ABB RAPID module: DecorationMovementV3

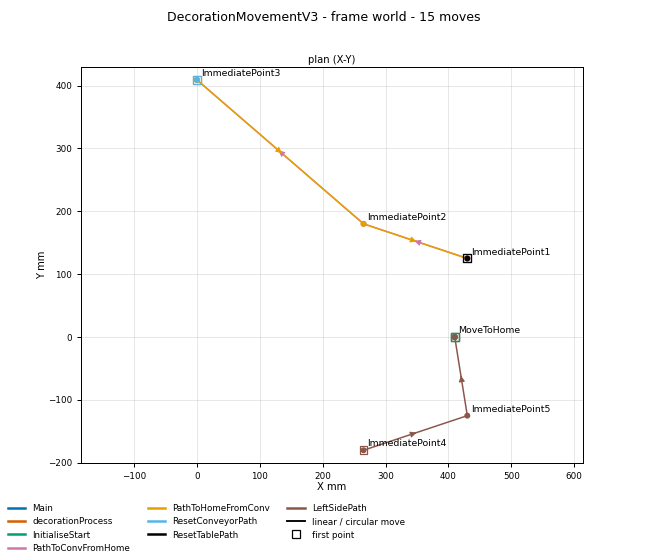
[picture p0: tool path of DecorationMovementV3 in frame world, 15 of 19 moves have a stored position in this frame; points joined in program order, loops and branches not executed]
MODULE DecorationFinal
!***************************************************************
! Decoration Movement Code for Robot
! Author: Dylan Dam z5115759
!***************************************************************


    ! Custom waypoints that I have selected
    CONST robtarget ImmediatePoint1:=[[430,125,450],[0,0,1,0],[0,-1,0,0],[9E+09,9E+09,9E+09,9E+09,9E+09,9E+09]];
    CONST robtarget ImmediatePoint2:=[[265,180,450],[0,0,1,0],[0,-1,0,0],[9E+09,9E+09,9E+09,9E+09,9E+09,9E+09]];
    CONST robtarget ImmediatePoint3:=[[0,409,450],[0,0,1,0],[1,-1,1,0],[9E+09,9E+09,9E+09,9E+09,9E+09,9E+09]];
    CONST robtarget ImmediatePoint4:=[[265,-180,450],[0,0,1,0],[1,-1,1,0],[9E+09,9E+09,9E+09,9E+09,9E+09,9E+09]];
    CONST robtarget ImmediatePoint5:=[[430,-125,450],[0,0,1,0],[1,-1,1,0],[9E+09,9E+09,9E+09,9E+09,9E+09,9E+09]];
    CONST robtarget MoveToHome:=[[410,0,450],[0,0,-1,0],[0,0,-1,0],[9E+09,9E+09,9E+09,9E+09,9E+09,9E+09]];
    ! Offset for the end-effector
    CONST num offSet := 75;
    !Dummy Array for Testing
    !CONST num qwirkleArray{4,7} := [[0,409,22.1,175,0,147,45],[0,409,22.1,548.6,0,147,0],[0,409,22.1,175,520,147,-45],[0,409,22.1,175,-300,147,-45]];
    CONST num qwirkleArray{1,7} := [[0,409,22.1,175,-50,147,-89]];

    PROC Main()
        MoveL MoveToHome,v1000,z100,tool0\WObj:=wobj0;
        decorationProcess qwirkleArray;
        MoveL MoveToHome,v1000,z100,tool0\WObj:=wobj0;
    ENDPROC

    PROC decorationProcess(num array{*,*})

        VAR num xStart;
        VAR num yStart;
        VAR num zStart;
        VAR num xEnd;
        VAR num yEnd;
        VAR num zEnd;
        VAR num orientation;
        VAR robtarget qwirkleLocation;
        VAR robtarget qwirklePlacement;

        FOR a FROM 1 TO Dim(array,1) DO
            ! This part reads in the first line.
            xEnd := array{a,1};
            yEnd := array{a,2};
            IF xEnd = 0 AND yEnd = 0 THEN
                ExitCycle;
            ENDIF
            !zStart := array{a,3}+offSet;
            zEnd := 147+offSet;
            xStart := array{a,4};
            yStart := array{a,5};
            zStart := 22.1+offSet;
            orientation := array{a,7};

            qwirklePlacement := [[xStart,yStart,zStart],[0,0,1,0],[0,0,0,0],[9E+09,9E+09,9E+09,9E+09,9E+09,9E+09]];
            qwirkleLocation :=[[xEnd,yEnd,zEnd],[0,0,1,0],[0,0,0,0],[9E+09,9E+09,9E+09,9E+09,9E+09,9E+09]];

            PathToConvFromHome;
            MoveL qwirkleLocation,v1000,z100,tool0\WObj:=wobj0;
            WaitTime 1;
            turnOnVacuum;
            turnOnGripper;
            ResetConveyorPath;
            PathToHomeFromConv;
            WaitTime 1;
            MoveL qwirklePlacement,v1000,z100,tool0\WObj:=wobj0;
            RotateTool orientation,qwirklePlacement;
            IF (yEnd < -400) THEN
                LeftSidePath;
            ELSE
                MoveL MoveToHome,v1000,z100,tool0\WObj:=wobj0;
            ENDIF

        ENDFOR

    ENDPROC

    PROC InitialiseStart()
        MoveL MoveToHome,v1000,z100,tool0\WObj:=wobj0;
    ENDPROC

    PROC PathToConvFromHome()
            MoveL ImmediatePoint1,v1000,z100,tool0\WObj:=wobj0;
            MoveL ImmediatePoint2,v1000,z100,tool0\WObj:=wobj0;
            MoveL ImmediatePoint3,v1000,z100,tool0\WObj:=wobj0;
    ENDPROC

    PROC PathToHomeFromConv()
        MoveL ImmediatePoint3,v1000,z100,tool0\WObj:=wobj0;
        MoveL ImmediatePoint2,v1000,z100,tool0\WObj:=wobj0;
        MoveL ImmediatePoint1,v1000,z100,tool0\WObj:=wobj0;
    ENDPROC
    PROC ResetConveyorPath()
        MoveL ImmediatePoint3,v1000,z100,tool0\WObj:=wobj0;
    ENDPROC
    PROC ResetTablePath()
        MoveL ImmediatePoint1,v1000,z100,tool0\WObj:=wobj0;
    ENDPROC

    PROC RotateTool(num Orientation,robtarget a)
        IF Orientation > 90 THEN
            Orientation := 90 - Orientation;
            MoveL RelTool(a,0,0,0,\Rz:= Orientation),v1000,fine,tool0\WObj:=wobj0;
            WaitTime 1;
            turnOffGripper;
            turnOffVacuum;
            WaitTime 1;
        ELSE
            MoveL RelTool(a,0,0,0,\Rz:= Orientation),v1000,fine,tool0\WObj:=wobj0;
            WaitTime 1;
            turnOffGripper;
            turnOffVacuum;
            WaitTime 1;
        ENDIF

    ENDPROC

    PROC LeftSidePath()

        MoveL ImmediatePoint4,v1000,z100,tool0\WObj:=wobj0;
        MoveL ImmediatePoint5,v1000,z100,tool0\WObj:=wobj0;
        MoveL MoveToHome,v1000,z100,tool0\WObj:=wobj0;


    ENDPROC

ENDMODULE
